FUNCTION_BLOCK T1_InsArray (* Basic Function Block Type *)
  (* Standard: 61499-2 *)
  (* Version 0.0, 2014-07-14, 4DIAC-IDE, 4DIAC-Consortium *)
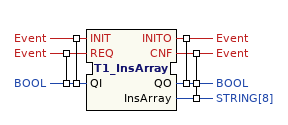
  EVENT_INPUT
    INIT WITH QI; (* Initialization Request *)
    REQ WITH QI; (* Normal Execution Request *)
  END_EVENT
  EVENT_OUTPUT
    INITO WITH QO; (* Initialization Confirm *)
    CNF WITH QO, InsArray; (* Execution Confirmation *)
  END_EVENT
  VAR_INPUT
    QI : BOOL; (* Input event qualifier *)
  END_VAR
  VAR_OUTPUT
    QO : BOOL; (* Output event qualifier *)
    InsArray : ARRAY [0..7] OF STRING := ['T4 D1','M6','G0 G17 G90 G94 F1000','S1000 M3','Z100','G88 G99 X0 Y0 Z2 I-10 D2 J35 B3 L0.5 H500 V50','G87 G98 X105 Y0 Z2 I-10 D2 J21 K28 M1 Q8  B3 L1 H480 V30','G0 G80 Z100'];
  END_VAR
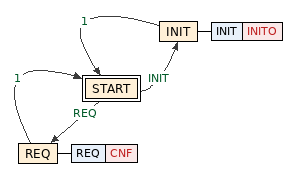
  EC_STATES
    START; (* Initial State *)
    INIT : INIT -> INITO; (* Initialization *)
    REQ : REQ -> CNF; (* Normal execution *)
  END_STATES
  EC_TRANSITIONS
    START TO INIT := INIT;
    INIT TO START := 1;
    START TO REQ := REQ;
    REQ TO START := 1;
  END_TRANSITIONS
  ALGORITHM INIT IN ST: (* Initialization algorithm *)

  END_ALGORITHM
  ALGORITHM REQ IN ST: (* Normally executed algorithm *)

  END_ALGORITHM
END_FUNCTION_BLOCK
